PROGRAM Stn2
VAR

	start2: BOOL;
	reset2: BOOL;

	Stn2ProcessFE: F_TRIG;
	Stn2ProcessRE: R_TRIG;
	bCutStn2ProcessHalt: BOOL;
	DoorClose2: R_TRIG;
	bStn2DoorClamp: BOOL;
END_VAR
VAR // added by the converter: edge detectors and wires of the graphical bodies
    _w1, _w2 : ANY;
END_VAR

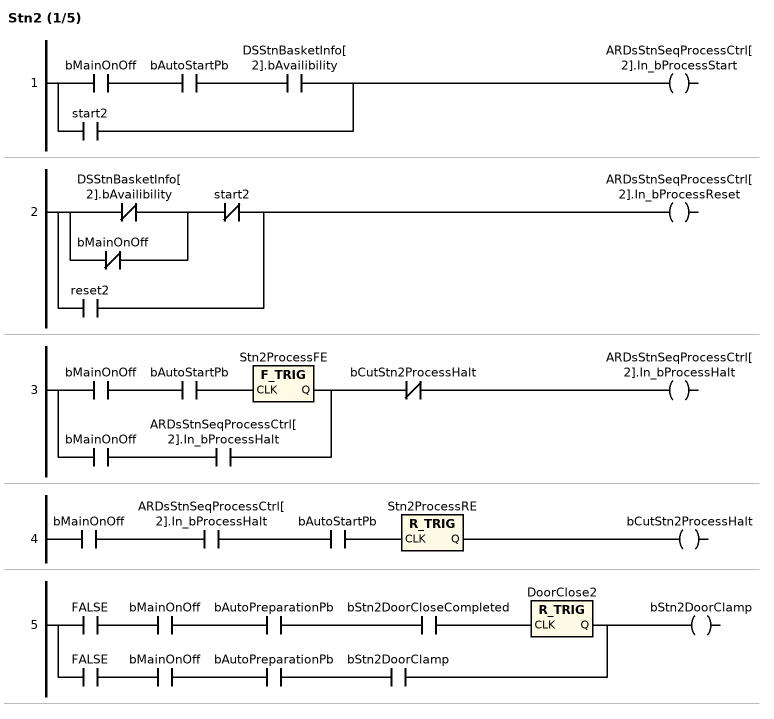
// NETWORK 1
ARDsStnSeqProcessCtrl[2].In_bProcessStart := bMainOnOff AND bAutoStartPb AND DSStnBasketInfo[2].bAvailibility OR start2;

// NETWORK 2
ARDsStnSeqProcessCtrl[2].In_bProcessReset := (NOT DSStnBasketInfo[2].bAvailibility OR NOT bMainOnOff) AND NOT start2 OR reset2;

// NETWORK 3
Stn2ProcessFE(CLK := bMainOnOff AND bAutoStartPb); // F_TRIG
ARDsStnSeqProcessCtrl[2].In_bProcessHalt := (Stn2ProcessFE.Q OR bMainOnOff AND ARDsStnSeqProcessCtrl[2].In_bProcessHalt) AND NOT bCutStn2ProcessHalt;

// NETWORK 4
Stn2ProcessRE(CLK := bMainOnOff AND ARDsStnSeqProcessCtrl[2].In_bProcessHalt AND bAutoStartPb); // R_TRIG
bCutStn2ProcessHalt := Stn2ProcessRE.Q;

// NETWORK 5
DoorClose2(CLK := (FALSE AND bMainOnOff AND bAutoPreparationPb) AND bStn2DoorCloseCompleted); // R_TRIG
bStn2DoorClamp := DoorClose2.Q OR (FALSE AND bMainOnOff AND bAutoPreparationPb) AND bStn2DoorClamp;

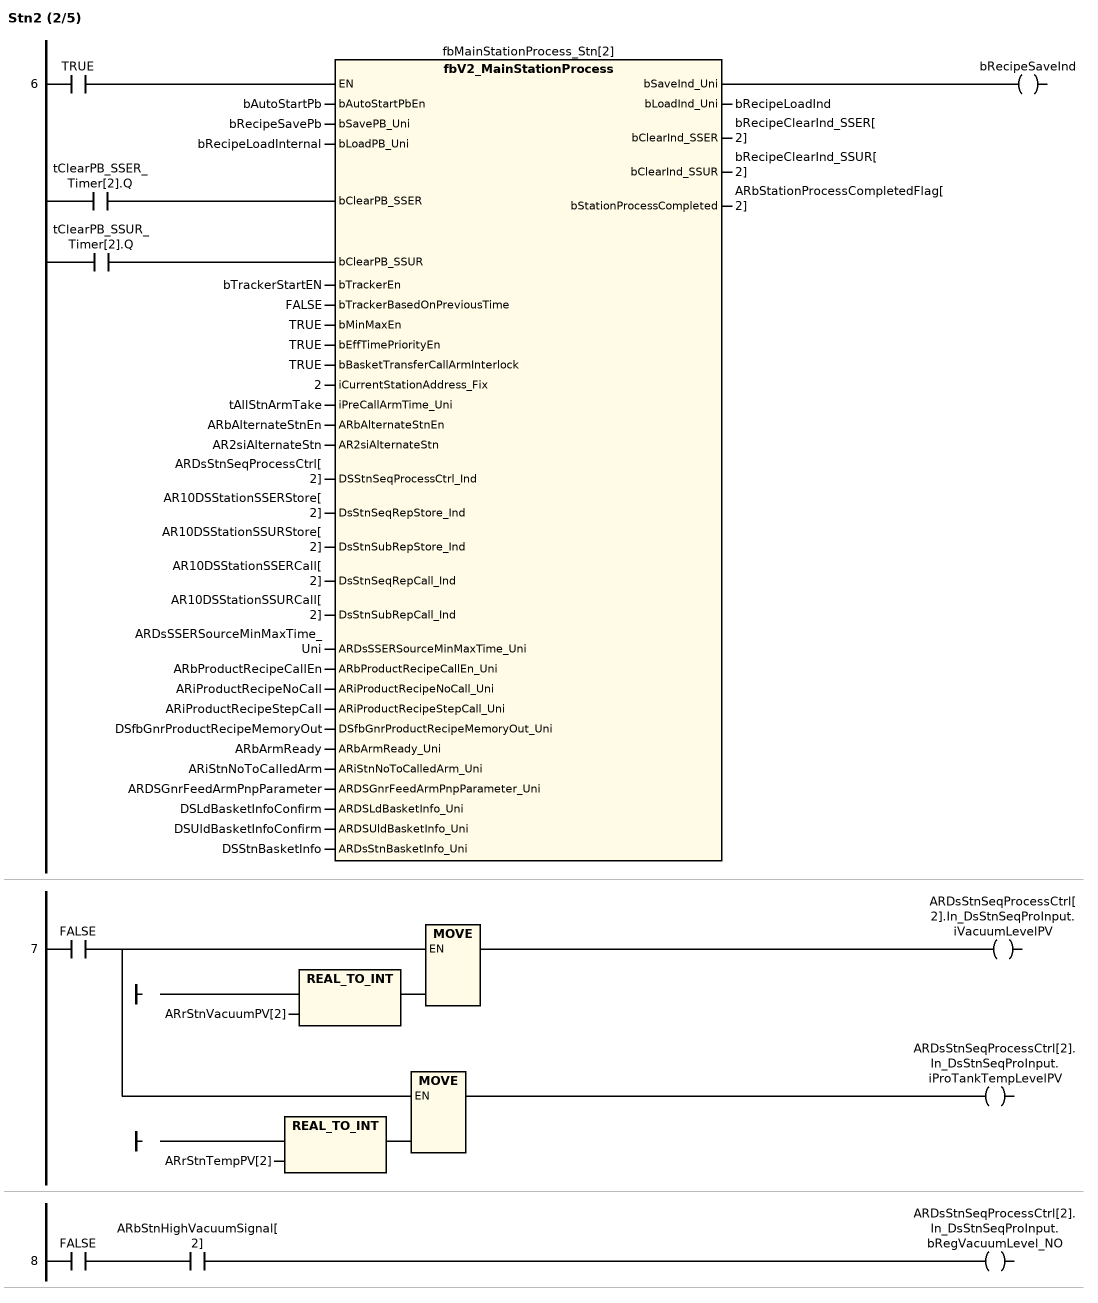
// NETWORK 6
fbMainStationProcess_Stn[2](
    bAutoStartPbEn := bAutoStartPb,
    bSavePB_Uni := bRecipeSavePb,
    bLoadPB_Uni := bRecipeLoadInternal,
    bClearPB_SSER := tClearPB_SSER_Timer[2].Q,
    bClearPB_SSUR := tClearPB_SSUR_Timer[2].Q,
    bTrackerEn := bTrackerStartEN,
    bTrackerBasedOnPreviousTime := FALSE,
    bMinMaxEn := TRUE,
    bEffTimePriorityEn := TRUE,
    bBasketTransferCallArmInterlock := TRUE,
    iCurrentStationAddress_Fix := 2,
    iPreCallArmTime_Uni := tAllStnArmTake,
    ARbAlternateStnEn := ARbAlternateStnEn,
    AR2siAlternateStn := AR2siAlternateStn,
    DSStnSeqProcessCtrl_Ind := ARDsStnSeqProcessCtrl[2],
    DsStnSeqRepStore_Ind := AR10DSStationSSERStore[2],
    DsStnSubRepStore_Ind := AR10DSStationSSURStore[2],
    DsStnSeqRepCall_Ind := AR10DSStationSSERCall[2],
    DsStnSubRepCall_Ind := AR10DSStationSSURCall[2],
    ARDsSSERSourceMinMaxTime_Uni := ARDsSSERSourceMinMaxTime_Uni,
    ARbProductRecipeCallEn_Uni := ARbProductRecipeCallEn,
    ARiProductRecipeNoCall_Uni := ARiProductRecipeNoCall,
    ARiProductRecipeStepCall_Uni := ARiProductRecipeStepCall,
    DSfbGnrProductRecipeMemoryOut_Uni := DSfbGnrProductRecipeMemoryOut,
    ARbArmReady_Uni := ARbArmReady,
    ARiStnNoToCalledArm_Uni := ARiStnNoToCalledArm,
    ARDSGnrFeedArmPnpParameter_Uni := ARDSGnrFeedArmPnpParameter,
    ARDSLdBasketInfo_Uni := DSLdBasketInfoConfirm,
    ARDSUldBasketInfo_Uni := DSUldBasketInfoConfirm,
    ARDsStnBasketInfo_Uni := DSStnBasketInfo,
    bLoadInd_Uni => bRecipeLoadInd,
    bClearInd_SSER => bRecipeClearInd_SSER[2],
    bClearInd_SSUR => bRecipeClearInd_SSUR[2],
    bStationProcessCompleted => ARbStationProcessCompletedFlag[2]); // fbV2_MainStationProcess
bRecipeSaveInd := fbMainStationProcess_Stn[2].bSaveInd_Uni;

// NETWORK 7
IF FALSE THEN _w1 := REAL_TO_INT(ARrStnVacuumPV[2]); END_IF
ARDsStnSeqProcessCtrl[2].In_DsStnSeqProInput.iVacuumLevelPV := _w1;
IF FALSE THEN _w2 := REAL_TO_INT(ARrStnTempPV[2]); END_IF
ARDsStnSeqProcessCtrl[2].In_DsStnSeqProInput.iProTankTempLevelPV := _w2;

// NETWORK 8
ARDsStnSeqProcessCtrl[2].In_DsStnSeqProInput.bRegVacuumLevel_NO := FALSE AND ARbStnHighVacuumSignal[2];

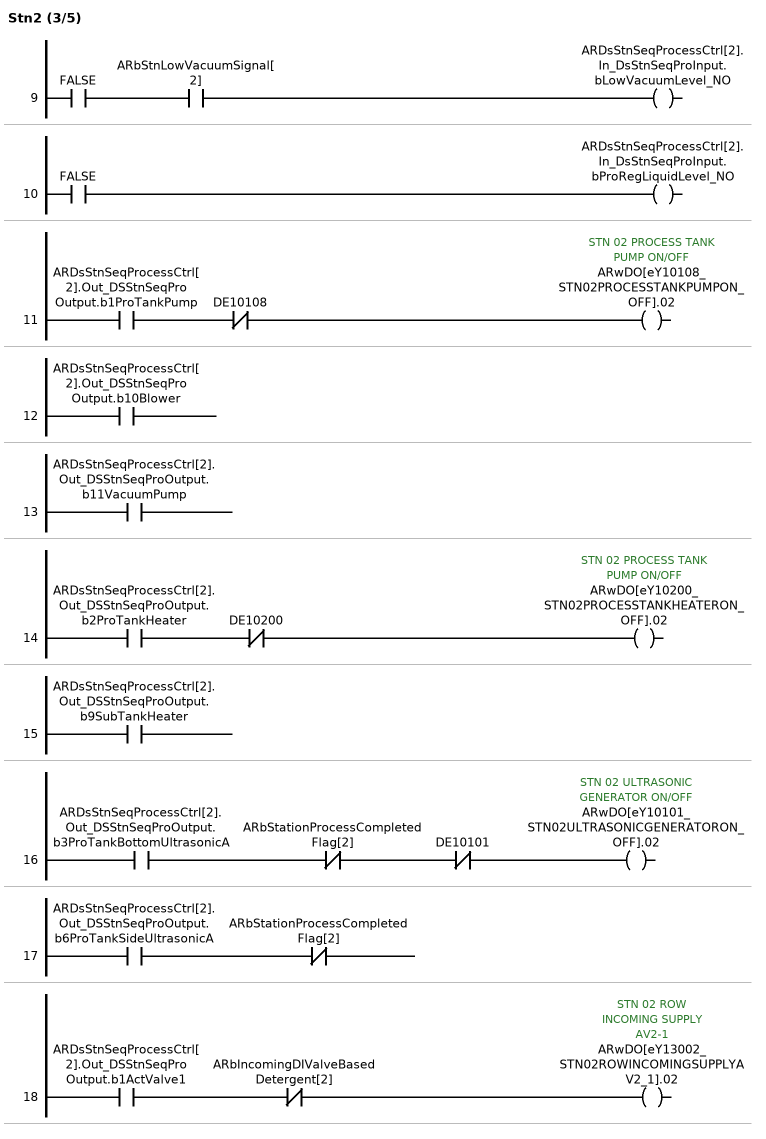
// NETWORK 9
ARDsStnSeqProcessCtrl[2].In_DsStnSeqProInput.bLowVacuumLevel_NO := FALSE AND ARbStnLowVacuumSignal[2];

// NETWORK 10
ARDsStnSeqProcessCtrl[2].In_DsStnSeqProInput.bProRegLiquidLevel_NO := FALSE;

// NETWORK 11
//   ARwDO[eY10108_STN02PROCESSTANKPUMPON_OFF].02: STN 02 PROCESS TANK PUMP ON/OFF
ARwDO[eY10108_STN02PROCESSTANKPUMPON_OFF].02 := ARDsStnSeqProcessCtrl[2].Out_DSStnSeqProOutput.b1ProTankPump AND NOT DE10108;

// NETWORK 12
(* ARDsStnSeqProcessCtrl[2].Out_DSStnSeqProOutput.b10Blower; not connected *)

// NETWORK 13
(* ARDsStnSeqProcessCtrl[2].Out_DSStnSeqProOutput.b11VacuumPump; not connected *)

// NETWORK 14
//   ARwDO[eY10200_STN02PROCESSTANKHEATERON_OFF].02: STN 02 PROCESS TANK PUMP ON/OFF
ARwDO[eY10200_STN02PROCESSTANKHEATERON_OFF].02 := ARDsStnSeqProcessCtrl[2].Out_DSStnSeqProOutput.b2ProTankHeater AND NOT DE10200;

// NETWORK 15
(* ARDsStnSeqProcessCtrl[2].Out_DSStnSeqProOutput.b9SubTankHeater; not connected *)

// NETWORK 16
//   ARwDO[eY10101_STN02ULTRASONICGENERATORON_OFF].02: STN 02 ULTRASONIC GENERATOR ON/OFF
ARwDO[eY10101_STN02ULTRASONICGENERATORON_OFF].02 := ARDsStnSeqProcessCtrl[2].Out_DSStnSeqProOutput.b3ProTankBottomUltrasonicA AND NOT ARbStationProcessCompletedFlag[2] AND NOT DE10101;

// NETWORK 17
(* ARDsStnSeqProcessCtrl[2].Out_DSStnSeqProOutput.b6ProTankSideUltrasonicA AND NOT ARbStationProcessCompletedFlag[2]; result not used *)

// NETWORK 18
//   ARwDO[eY13002_STN02ROWINCOMINGSUPPLYAV2_1].02: STN 02 ROW INCOMING SUPPLY AV2-1
ARwDO[eY13002_STN02ROWINCOMINGSUPPLYAV2_1].02 := ARDsStnSeqProcessCtrl[2].Out_DSStnSeqProOutput.b1ActValve1 AND NOT ARbIncomingDIValveBasedDetergent[2];

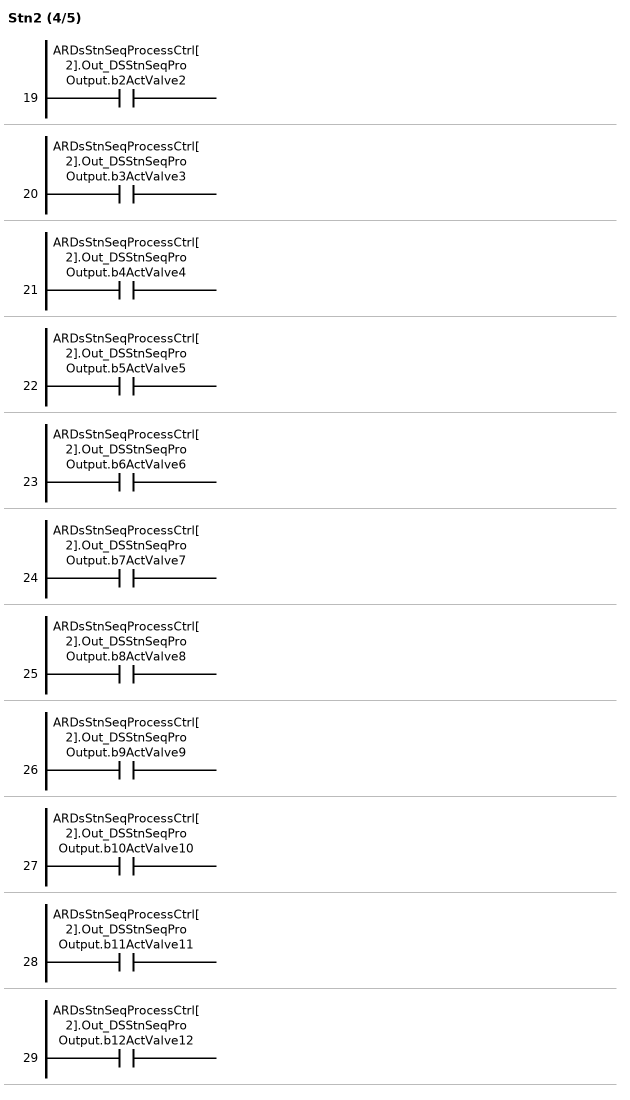
// NETWORK 19
(* ARDsStnSeqProcessCtrl[2].Out_DSStnSeqProOutput.b2ActValve2; not connected *)

// NETWORK 20
(* ARDsStnSeqProcessCtrl[2].Out_DSStnSeqProOutput.b3ActValve3; not connected *)

// NETWORK 21
(* ARDsStnSeqProcessCtrl[2].Out_DSStnSeqProOutput.b4ActValve4; not connected *)

// NETWORK 22
(* ARDsStnSeqProcessCtrl[2].Out_DSStnSeqProOutput.b5ActValve5; not connected *)

// NETWORK 23
(* ARDsStnSeqProcessCtrl[2].Out_DSStnSeqProOutput.b6ActValve6; not connected *)

// NETWORK 24
(* ARDsStnSeqProcessCtrl[2].Out_DSStnSeqProOutput.b7ActValve7; not connected *)

// NETWORK 25
(* ARDsStnSeqProcessCtrl[2].Out_DSStnSeqProOutput.b8ActValve8; not connected *)

// NETWORK 26
(* ARDsStnSeqProcessCtrl[2].Out_DSStnSeqProOutput.b9ActValve9; not connected *)

// NETWORK 27
(* ARDsStnSeqProcessCtrl[2].Out_DSStnSeqProOutput.b10ActValve10; not connected *)

// NETWORK 28
(* ARDsStnSeqProcessCtrl[2].Out_DSStnSeqProOutput.b11ActValve11; not connected *)

// NETWORK 29
(* ARDsStnSeqProcessCtrl[2].Out_DSStnSeqProOutput.b12ActValve12; not connected *)

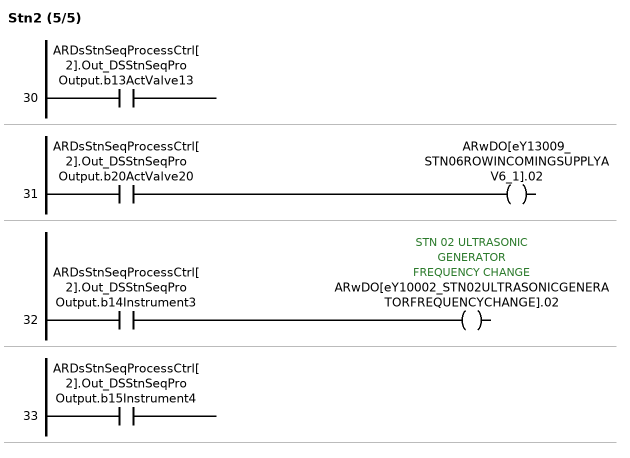
// NETWORK 30
(* ARDsStnSeqProcessCtrl[2].Out_DSStnSeqProOutput.b13ActValve13; not connected *)

// NETWORK 31
ARwDO[eY13009_STN06ROWINCOMINGSUPPLYAV6_1].02 := ARDsStnSeqProcessCtrl[2].Out_DSStnSeqProOutput.b20ActValve20;

// NETWORK 32
//   ARwDO[eY10002_STN02ULTRASONICGENERATORFREQUENCYCHANGE].02: STN 02 ULTRASONIC GENERATOR FREQUENCY CHANGE
ARwDO[eY10002_STN02ULTRASONICGENERATORFREQUENCYCHANGE].02 := ARDsStnSeqProcessCtrl[2].Out_DSStnSeqProOutput.b14Instrument3;

// NETWORK 33
(* ARDsStnSeqProcessCtrl[2].Out_DSStnSeqProOutput.b15Instrument4; not connected *)

END_PROGRAM

(* stored: Version 1.1.0.1, ProductVersion 3.1.4024.12
   POU Stn2: Id {80a7b387-4324-432d-9303-8e8fb22d48d8}, SpecialFunc None *)
